Staubli VAL3: del.pgx

public program del(num x_nIndex)
begin
  //delete(saveAxis[x_nIndex])
  if size(nSaveaxis)>1
    $ddel(nSaveaxis,x_nIndex)
    $ddel(nSaveaxis1,x_nIndex)
    $ddel(sSaveaxis,x_nIndex)
    $ddel(nVelocity,x_nIndex)
  endIf
end
